Fanuc TP program (LS listing): __main.ls

/PROG  __MAIN
/ATTR
OWNER		= MNEDITOR;
COMMENT		= "MAIN PROG CALL";
PROG_SIZE	= 291;
CREATE		= DATE 24-11-11  TIME 10:41:58;
MODIFIED	= DATE 24-11-11  TIME 10:41:58;
FILE_NAME	= ;
VERSION		= 0;
LINE_COUNT	= 8;
MEMORY_SIZE	= 779;
PROTECT		= READ_WRITE;
TCD:  STACK_SIZE	= 0,
      TASK_PRIORITY	= 50,
      TIME_SLICE	= 0,
      BUSY_LAMP_OFF	= 0,
      ABORT_REQUEST	= 0,
      PAUSE_REQUEST	= 0;
DEFAULT_GROUP	= 1,*,*,*,*;
CONTROL_CODE	= 00000000 00000000;
LOCAL_REGISTERS	= 0,0,0;
/APPL

AUTO_SINGULARITY_HEADER;
  ENABLE_SINGULARITY_AVOIDANCE   : TRUE;
/MN
   1:  LBL[100] ;
   2:  DO[1:OFF:Auto Mode Echo]=OFF ;
   3:  DO[2:OFF:Running]=OFF ;
   4:   ;
   5:  IF (DI[1:ON :Auto Mode]),CALL __AUTO ;
   6:  IF (!DI[1:ON :Auto Mode]),CALL __MANUAL ;
   7:  WAIT    .25(sec) ;
   8:  JMP LBL[100] ;
/POS
/END
